	    //Übertragung in Melde-DB
	    "FC63_DB_Copy"(DB_src := 80,
	                   DB_src_offs := 96,
	                   DB_dest := 100,
	                   DB_dest_offs := 64,
	                   count := 34);
	    //div. Messwerte
	    "ZEN_MW".BB_G1_KS_Druck_Netz := INT_TO_REAL("DB80_Peri_EA".Kaeser_G1.E.Druck_Netz) / 1.0;
	    "ZEN_MW".BB_G1_KS_Temp_Verdicht := INT_TO_REAL("DB80_Peri_EA".Kaeser_G1.E.Temp_Verdicht) / 10.0;
	    "ZEN_MW".BB_G1_KS_Temp_Schallhaube := INT_TO_REAL("DB80_Peri_EA".Kaeser_G1.E.Temp_Schallhaube) / 10.0;
	    "ZEN_MW".BB_G1_KS_Temp_Ansaug := INT_TO_REAL("DB80_Peri_EA".Kaeser_G1.E.Temp_Ansaug) / 10.0;
	    "ZEN_MW".BB_G1_KS_Temp_Oel := INT_TO_REAL("DB80_Peri_EA".Kaeser_G1.E.Temp_Oel) / 10.0;
	    "ZEN_MW".BB_G1_KS_Temp_Wicklung := INT_TO_REAL("DB80_Peri_EA".Kaeser_G1.E.Temp_Wicklung) / 10.0;
	    "ZEN_MW".BB_G1_KS_Volumenstrom := INT_TO_REAL("DB80_Peri_EA".Kaeser_G1.E.Volumenstrom) * 6.0;
	    "ZEN_MW".BB_G1_KS_Motorfrequenz := INT_TO_REAL("DB80_Peri_EA".Kaeser_G1.E.Motorfrequenz) / 1.0;
	    "ZEN_MW".BB_G1_KS_Motordrehzahl := UINT_TO_REAL("DB80_Peri_EA".Kaeser_G1.E.Motordrehzahl) / 1.0;
	    "ZEN_MW".BB_G1_KS_Blockdrehzahl := UINT_TO_REAL("DB80_Peri_EA".Kaeser_G1.E.Blockdrehzahl) / 1.0;
	END_IF;
	//dezentrale Peripherie Kaeser Gebläse 2 - Teilnehmer 7
	IF "DB91_DP_aktiv".Tln[7] THEN
	    "FC63_DB_Copy"(DB_src := 0,
	                   DB_src_offs := 1200,
	                   DB_dest := 80,
	                   DB_dest_offs := 296,
	                   count := 128);
	    "FC63_DB_Copy"(DB_src := 80,
	                   DB_src_offs := 424,
	                   DB_dest := 0,
	                   DB_dest_offs := 1200,
	                   count := 64);

	    //Übertragung in Melde-DB
	    "FC63_DB_Copy"(DB_src := 80,
	                   DB_src_offs := 296,
	                   DB_dest := 100,
	                   DB_dest_offs := 98,
	                   count := 34);
	    //div. Messwerte
	    "ZEN_MW".BB_G2_KS_Druck_Netz := INT_TO_REAL("DB80_Peri_EA".Kaeser_G2.E.Druck_Netz) / 1.0;
	    "ZEN_MW".BB_G2_KS_Temp_Verdicht := INT_TO_REAL("DB80_Peri_EA".Kaeser_G2.E.Temp_Verdicht) / 10.0;
	    "ZEN_MW".BB_G2_KS_Temp_Schallhaube := INT_TO_REAL("DB80_Peri_EA".Kaeser_G2.E.Temp_Schallhaube) / 10.0;
	    "ZEN_MW".BB_G2_KS_Temp_Ansaug := INT_TO_REAL("DB80_Peri_EA".Kaeser_G2.E.Temp_Ansaug) / 10.0;
	    "ZEN_MW".BB_G2_KS_Temp_Oel := INT_TO_REAL("DB80_Peri_EA".Kaeser_G2.E.Temp_Oel) / 10.0;
	    "ZEN_MW".BB_G2_KS_Temp_Wicklung := INT_TO_REAL("DB80_Peri_EA".Kaeser_G2.E.Temp_Wicklung) / 10.0;
	    "ZEN_MW".BB_G2_KS_Volumenstrom := INT_TO_REAL("DB80_Peri_EA".Kaeser_G2.E.Volumenstrom) * 6.0;
	    "ZEN_MW".BB_G2_KS_Motorfrequenz := INT_TO_REAL("DB80_Peri_EA".Kaeser_G2.E.Motorfrequenz) / 1.0;
	    "ZEN_MW".BB_G2_KS_Motordrehzahl := UINT_TO_REAL("DB80_Peri_EA".Kaeser_G2.E.Motordrehzahl) / 1.0;
	    "ZEN_MW".BB_G2_KS_Blockdrehzahl := UINT_TO_REAL("DB80_Peri_EA".Kaeser_G2.E.Blockdrehzahl) / 1.0;

	END_IF;
	//dezentrale Peripherie Kaeser Gebläse 3 - Teilnehmer 8
	IF "DB91_DP_aktiv".Tln[8] THEN
	    "FC63_DB_Copy"(DB_src := 0,
	                   DB_src_offs := 1400,
	                   DB_dest := 80,
	                   DB_dest_offs := 496,
	                   count := 128);
	    "FC63_DB_Copy"(DB_src := 80,
	                   DB_src_offs := 624,
	                   DB_dest := 0,
	                   DB_dest_offs := 1400,
	                   count := 64);

	    //Übertragung in Melde-DB
	    "FC63_DB_Copy"(DB_src := 80,
	                   DB_src_offs := 496,
	                   DB_dest := 100,
	                   DB_dest_offs := 132,
	                   count := 34);
	    //div. Messwerte
	    "ZEN_MW".BB_G3_KS_Druck_Netz := INT_TO_REAL("DB80_Peri_EA".Kaeser_G3.E.Druck_Netz) / 1.0;
	    "ZEN_MW".BB_G3_KS_Temp_Verdicht := INT_TO_REAL("DB80_Peri_EA".Kaeser_G3.E.Temp_Verdicht) / 10.0;
	    "ZEN_MW".BB_G3_KS_Temp_Schallhaube := INT_TO_REAL("DB80_Peri_EA".Kaeser_G3.E.Temp_Schallhaube) / 10.0;
	    "ZEN_MW".BB_G3_KS_Temp_Ansaug := INT_TO_REAL("DB80_Peri_EA".Kaeser_G3.E.Temp_Ansaug) / 10.0;
	    "ZEN_MW".BB_G3_KS_Temp_Oel := INT_TO_REAL("DB80_Peri_EA".Kaeser_G3.E.Temp_Oel) / 10.0;
	    "ZEN_MW".BB_G3_KS_Temp_Wicklung := INT_TO_REAL("DB80_Peri_EA".Kaeser_G3.E.Temp_Wicklung) / 10.0;
	    "ZEN_MW".BB_G3_KS_Volumenstrom := INT_TO_REAL("DB80_Peri_EA".Kaeser_G3.E.Volumenstrom)*6.0;
	    "ZEN_MW".BB_G3_KS_Motorfrequenz := INT_TO_REAL("DB80_Peri_EA".Kaeser_G3.E.Motorfrequenz) / 1.0;
	    "ZEN_MW".BB_G3_KS_Motordrehzahl := UINT_TO_REAL("DB80_Peri_EA".Kaeser_G3.E.Motordrehzahl) / 1.0;
	    "ZEN_MW".BB_G3_KS_Blockdrehzahl := UINT_TO_REAL("DB80_Peri_EA".Kaeser_G3.E.Blockdrehzahl) / 1.0;

	END_IF;


	"ZEN_Meld".ZEN_DiagKom_DP_BF3 := NOT "DB91_DP_aktiv".Tln[3];
	"ZEN_Meld".ZEN_DiagKom_DP_BF4 := NOT "DB91_DP_aktiv".Tln[4];
	"ZEN_Meld".ZEN_DiagKom_DP_BF5 := NOT "DB91_DP_aktiv".Tln[5];
	"ZEN_Meld".ZEN_DiagKom_DP_BF6 := NOT "DB91_DP_aktiv".Tln[6];
	"ZEN_Meld".ZEN_DiagKom_DP_BF7 := NOT "DB91_DP_aktiv".Tln[7];
	"ZEN_Meld".ZEN_DiagKom_DP_BF8 := NOT "DB91_DP_aktiv".Tln[8];
	"ZEN_Meld".ZEN_DiagKom_DP_BF10 := NOT "DB91_DP_aktiv".Tln[10];

	//Meldungen für OP
	//
	IF 1 THEN

	    "DB92_OP_Data".Msg_B0[0].%X0 := "ZEN_Meld".E_Zulauf_AR_P1_St;
	    "DB92_OP_Data".Msg_B0[0].%X1 := "ZEN_Meld".E_Zulauf_AR_SS;
	    "DB92_OP_Data".Msg_B0[0].%X2 := "ZEN_Meld".E_Zulauf_AR_P2_St;
	    "DB92_OP_Data".Msg_B0[0].%X3 := "ZEN_Meld".E_Zulauf_AR_HW;
	    "DB92_OP_Data".Msg_B0[0].%X4 := "ZEN_Meld".E_Zulauf_AR_Niv_St;
	    "DB92_OP_Data".Msg_B0[0].%X5 := "ZEN_Meld".E_Zulauf_AR_DF_St;
	    "DB92_OP_Data".Msg_B0[0].%X6 := "ZEN_Meld".E_Ablauf_pH_St;
	    "DB92_OP_Data".Msg_B0[0].%X7 := "ZEN_Meld".E_Ablauf_O2_St;
	    "DB92_OP_Data".Msg_B0[0].%X8 := "ZEN_Meld".E_Ablauf_DF_St;
	    "DB92_OP_Data".Msg_B0[0].%X9 := "ZEN_Meld".E_NSHV_SS1_St;
	    "DB92_OP_Data".Msg_B0[0].%X10 := "ZEN_Meld".E_NSHV_SS2_St;
	    "DB92_OP_Data".Msg_B0[0].%X11 := "ZEN_Meld".E_NSHV_N02_AF_St;
	    "DB92_OP_Data".Msg_B0[0].%X12 := "ZEN_Meld".E_NSHV_N03_AF_St;
	    "DB92_OP_Data".Msg_B0[0].%X13 := "ZEN_Meld".E_NSHV_N04_AF_St;
	    "DB92_OP_Data".Msg_B0[0].%X14 := "ZEN_Meld".E_NSHV_LS_Aus;
	    "DB92_OP_Data".Msg_B0[0].%X15 := "ZEN_Meld".E_NSHV_LS_St;
	    "DB92_OP_Data".Msg_B0[1].%X0 := "ZEN_Meld".E_NSHV_NA;
	    "DB92_OP_Data".Msg_B0[1].%X1 := "ZEN_Meld".E_BB_G1_St;
	    "DB92_OP_Data".Msg_B0[1].%X2 := "ZEN_Meld".E_BB_G1_AF_St;
	    "DB92_OP_Data".Msg_B0[1].%X3 := "ZEN_Meld".E_BB_SHL_G1_St;
	    "DB92_OP_Data".Msg_B0[1].%X4 := "ZEN_Meld".E_BB_G2_St;
	    "DB92_OP_Data".Msg_B0[1].%X5 := "ZEN_Meld".E_BB_G2_AF_St;
	    "DB92_OP_Data".Msg_B0[1].%X6 := "ZEN_Meld".E_BB_SHL_G2_St;
	    "DB92_OP_Data".Msg_B0[1].%X7 := "ZEN_Meld".E_BB_G3_St;
	    "DB92_OP_Data".Msg_B0[1].%X8 := "ZEN_Meld".E_BB_G3_AF_St;
	    "DB92_OP_Data".Msg_B0[1].%X9 := "ZEN_Meld".E_BB_SHL_G3_St;
	    "DB92_OP_Data".Msg_B0[1].%X10 := "ZEN_Meld".E_BB_AV_St;
	    "DB92_OP_Data".Msg_B0[1].%X11 := "ZEN_Meld".E_BB_AV_AF_St;
	    "DB92_OP_Data".Msg_B0[1].%X12 := "ZEN_Meld".E_BB_RT;
	    "DB92_OP_Data".Msg_B0[1].%X13 := "ZEN_Meld".E_BB1_SR_K_St;
	    "DB92_OP_Data".Msg_B0[1].%X14 := "ZEN_Meld".E_BB1_SR_K_AF_St;
	    "DB92_OP_Data".Msg_B0[1].%X15 := "ZEN_Meld".E_BB_LS1_St;
	    "DB92_OP_Data".Msg_B0[2].%X0 := "ZEN_Meld".E_BB_LS1_AF_St;
	    "DB92_OP_Data".Msg_B0[2].%X1 := "ZEN_Meld".E_BB_LS2_St;
	    "DB92_OP_Data".Msg_B0[2].%X2 := "ZEN_Meld".E_BB_LS2_AF_St;
	    "DB92_OP_Data".Msg_B0[2].%X3 := "ZEN_Meld".E_BB1_RZP1_St;
	    "DB92_OP_Data".Msg_B0[2].%X4 := "ZEN_Meld".E_BB1_RZP1_AF_St;
	    "DB92_OP_Data".Msg_B0[2].%X5 := "ZEN_Meld".E_BB1_RZP2_St;
	    "DB92_OP_Data".Msg_B0[2].%X6 := "ZEN_Meld".E_BB1_RZP2_AF_St;
	    "DB92_OP_Data".Msg_B0[2].%X7 := "ZEN_Meld".E_BB1_UeSP_St;
	    "DB92_OP_Data".Msg_B0[2].%X8 := "ZEN_Meld".E_BB1_UeSP_AF_St;
	    "DB92_OP_Data".Msg_B0[2].%X9 := "ZEN_Meld".E_BB1_AS1_St;
	    "DB92_OP_Data".Msg_B0[2].%X10 := "ZEN_Meld".E_BB1_AS1_AF_St;
	    "DB92_OP_Data".Msg_B0[2].%X11 := "ZEN_Meld".E_BB1_AS2_St;
	    "DB92_OP_Data".Msg_B0[2].%X12 := "ZEN_Meld".E_BB1_AS2_AF_St;
	    "DB92_OP_Data".Msg_B0[2].%X13 := "ZEN_Meld".E_BB1_SR1_AF_St;
	    "DB92_OP_Data".Msg_B0[2].%X14 := "ZEN_Meld".E_BB1_SR2_AF_St;
	    "DB92_OP_Data".Msg_B0[2].%X15 := "ZEN_Meld".E_BB1_O2_St;
	    "DB92_OP_Data".Msg_B0[3].%X0 := "ZEN_Meld".E_BB1_DF_St;
	    "DB92_OP_Data".Msg_B0[3].%X1 := "ZEN_Meld".E_BB2_RZP1_St;
	    "DB92_OP_Data".Msg_B0[3].%X2 := "ZEN_Meld".E_BB2_RZP1_AF_St;
	    "DB92_OP_Data".Msg_B0[3].%X3 := "ZEN_Meld".E_BB2_RZP2_St;
	    "DB92_OP_Data".Msg_B0[3].%X4 := "ZEN_Meld".E_BB2_RZP2_AF_St;
	    "DB92_OP_Data".Msg_B0[3].%X5 := "ZEN_Meld".E_BB2_UeSP_St;
	    "DB92_OP_Data".Msg_B0[3].%X6 := "ZEN_Meld".E_BB2_UeSP_AF_St;
	    "DB92_OP_Data".Msg_B0[3].%X7 := "ZEN_Meld".E_BB2_AS1_St;
	    "DB92_OP_Data".Msg_B0[3].%X8 := "ZEN_Meld".E_BB2_AS1_AF_St;
	    "DB92_OP_Data".Msg_B0[3].%X9 := "ZEN_Meld".E_BB2_AS2_St;
	    "DB92_OP_Data".Msg_B0[3].%X10 := "ZEN_Meld".E_BB2_AS2_AF_St;
	    "DB92_OP_Data".Msg_B0[3].%X11 := "ZEN_Meld".E_BB2_SR1_AF_St;
	    "DB92_OP_Data".Msg_B0[3].%X12 := "ZEN_Meld".E_BB2_SR2_AF_St;
	    "DB92_OP_Data".Msg_B0[3].%X13 := "ZEN_Meld".E_BB2_O2_St;
	    "DB92_OP_Data".Msg_B0[3].%X14 := "ZEN_Meld".E_BB2_DF_St;
	    "DB92_OP_Data".Msg_B0[3].%X15 := "ZEN_Meld".E_BB2_SR_K_St;
	    "DB92_OP_Data".Msg_B0[4].%X0 := "ZEN_Meld".E_BB2_SR_K_AF_St;
	    "DB92_OP_Data".Msg_B0[4].%X1 := "ZEN_Meld".E_Zulauf_RA_SA_St;
	    "DB92_OP_Data".Msg_B0[4].%X2 := "ZEN_Meld".E_Zulauf_RA_HZS_St;
	    "DB92_OP_Data".Msg_B0[4].%X3 := "ZEN_Meld".E_Zulauf_RA_VKS_St;
	    "DB92_OP_Data".Msg_B0[4].%X4 := "ZEN_Meld".E_Zulauf_RA_V_St;
	    "DB92_OP_Data".Msg_B0[4].%X5 := "ZEN_Meld".E_Zulauf_RA_RP_St;
	    "DB92_OP_Data".Msg_B0[4].%X6 := "ZEN_Meld".E_Zulauf_RA_FP_St;
	    "DB92_OP_Data".Msg_B0[4].%X7 := "ZEN_Meld".E_Zulauf_RA_24V_St;
	    "DB92_OP_Data".Msg_B0[4].%X8 := "ZEN_Meld".E_Zulauf_RA_US_St;
	    "DB92_OP_Data".Msg_B0[4].%X9 := "ZEN_Meld".E_Zulauf_RA_230V_St;
	    "DB92_OP_Data".Msg_B0[4].%X10 := "ZEN_Meld".E_Zulauf_DF_St;
	    "DB92_OP_Data".Msg_B0[4].%X11 := "ZEN_Meld".E_Zulauf_Niv_St;
	    "DB92_OP_Data".Msg_B0[4].%X12 := "ZEN_Meld".E_Verteiler_pH_St;
	    "DB92_OP_Data".Msg_B0[4].%X13 := "ZEN_Meld".E_Zulauf_AS_St;
	    "DB92_OP_Data".Msg_B0[4].%X14 := "ZEN_Meld".E_Zulauf_AS_AF_St;
	    "DB92_OP_Data".Msg_B0[4].%X15 := "ZEN_Meld".E_Schlamm_BP_St;
	    "DB92_OP_Data".Msg_B0[5].%X0 := "ZEN_Meld".E_Schlamm_BP_AF_St;
	    "DB92_OP_Data".Msg_B0[5].%X1 := "ZEN_Meld".E_Truebwasser_P1_St;
	    "DB92_OP_Data".Msg_B0[5].%X2 := "ZEN_Meld".E_Truebwasser_P1_AF_St;
	    "DB92_OP_Data".Msg_B0[5].%X3 := "ZEN_Meld".E_Truebwasser_P2_St;
	    "DB92_OP_Data".Msg_B0[5].%X4 := "ZEN_Meld".E_Truebwasser_P2_AF_St;
	    "DB92_OP_Data".Msg_B0[5].%X5 := "ZEN_Meld".E_Schlamm_AS_St;
	    "DB92_OP_Data".Msg_B0[5].%X6 := "ZEN_Meld".E_Schlamm_AS_AF_St;
	    "DB92_OP_Data".Msg_B0[5].%X7 := "ZEN_Meld".E_Schlamm_Besch_DF_St;
	    "DB92_OP_Data".Msg_B0[5].%X8 := "ZEN_Meld".E_Truebwasser_Niv_St;
	    "DB92_OP_Data".Msg_B0[5].%X9 := "ZEN_Meld".E_Truebwasser_DF_St;
	    "DB92_OP_Data".Msg_B0[5].%X10 := "ZEN_Meld".ZEN_DiagKom_IEC;
	    "DB92_OP_Data".Msg_B0[5].%X11 := "ZEN_Meld".ZEN_DiagKom_DP_BF3;
	    "DB92_OP_Data".Msg_B0[5].%X12 := "ZEN_Meld".ZEN_DiagKom_DP_BF4;
	    "DB92_OP_Data".Msg_B0[5].%X13 := "ZEN_Meld".ZEN_ObjS_Alarm;
	    "DB92_OP_Data".Msg_B0[5].%X14 := "ZEN_Meld".ZEN_ObjS_unscharf;
	    "DB92_OP_Data".Msg_B0[5].%X15 := "ZEN_Meld".ZEN_NA_res;
	    "DB92_OP_Data".Msg_B0[6].%X0 := "ZEN_Meld".Biocos1_Auto_Bel_O2_St;
	    "DB92_OP_Data".Msg_B0[6].%X1 := "ZEN_Meld".Biocos1_Auto_Bel_O2_min;
	    "DB92_OP_Data".Msg_B0[6].%X2 := "ZEN_Meld".Biocos1_Auto_UeSS_Menge_St;
	    "DB92_OP_Data".Msg_B0[6].%X3 := "ZEN_Meld".Biocos2_Auto_Bel_O2_St;
	    "DB92_OP_Data".Msg_B0[6].%X4 := "ZEN_Meld".Biocos2_Auto_Bel_O2_min;
	    "DB92_OP_Data".Msg_B0[6].%X5 := "ZEN_Meld".Biocos2_Auto_UeSS_Menge_St;
	    "DB92_OP_Data".Msg_B0[6].%X6 := "ZEN_Meld".Zulauf_PW_Auto_DF_max;
	    "DB92_OP_Data".Msg_B0[6].%X7 := "ZEN_Meld".Zulauf_PW_Auto_Niv_max;
	    "DB92_OP_Data".Msg_B0[6].%X8 := "ZEN_Meld".Zulauf_PW_Auto_Niv_AS;
	    "DB92_OP_Data".Msg_B0[6].%X9 := "ZEN_Meld".Zulauf_PW_Auto_Frg_Aus;
	    "DB92_OP_Data".Msg_B0[6].%X10 := "ZEN_Meld".Zulauf_RA_SA_Stillst;
	    "DB92_OP_Data".Msg_B0[6].%X11 := "ZEN_Meld".Schlamm_Besch_Auto_Zt_max;
	    "DB92_OP_Data".Msg_B0[6].%X12 := "DB104_Antriebe_Meld".BB_G1.Stoerung.Wa_EZ;
	    "DB92_OP_Data".Msg_B0[6].%X13 := "DB104_Antriebe_Meld".BB_G1.Stoerung.Wa_Wart;
	    "DB92_OP_Data".Msg_B0[6].%X14 := "DB104_Antriebe_Meld".BB_G2.Stoerung.Wa_EZ;
	    "DB92_OP_Data".Msg_B0[6].%X15 := "DB104_Antriebe_Meld".BB_G2.Stoerung.Wa_Wart;
	    "DB92_OP_Data".Msg_B0[7].%X0 := "DB104_Antriebe_Meld".BB_G3.Stoerung.Wa_EZ;
	    "DB92_OP_Data".Msg_B0[7].%X1 := "DB104_Antriebe_Meld".BB_G3.Stoerung.Wa_Wart;
	    "DB92_OP_Data".Msg_B0[7].%X2 := "DB104_Antriebe_Meld".BB_SHL_G1.Stoerung.Wa_EZ;
	    "DB92_OP_Data".Msg_B0[7].%X3 := "DB104_Antriebe_Meld".BB_SHL_G1.Stoerung.Wa_Wart;
	    "DB92_OP_Data".Msg_B0[7].%X4 := "DB104_Antriebe_Meld".BB_SHL_G2.Stoerung.Wa_EZ;
	    "DB92_OP_Data".Msg_B0[7].%X5 := "DB104_Antriebe_Meld".BB_SHL_G2.Stoerung.Wa_Wart;
	    "DB92_OP_Data".Msg_B0[7].%X6 := "DB104_Antriebe_Meld".BB_SHL_G3.Stoerung.Wa_EZ;
	    "DB92_OP_Data".Msg_B0[7].%X7 := "DB104_Antriebe_Meld".BB_SHL_G3.Stoerung.Wa_Wart;
	    "DB92_OP_Data".Msg_B0[7].%X8 := "DB104_Antriebe_Meld".BB_AV.Stoerung.Wa_EZ;
	    "DB92_OP_Data".Msg_B0[7].%X9 := "DB104_Antriebe_Meld".BB_AV.Stoerung.Wa_Wart;
	    "DB92_OP_Data".Msg_B0[7].%X10 := "DB104_Antriebe_Meld".BB_LS1.Stoerung.Wa_EZ;
	    "DB92_OP_Data".Msg_B0[7].%X11 := "DB104_Antriebe_Meld".BB_LS1.Stoerung.Wa_Wart;
	    "DB92_OP_Data".Msg_B0[7].%X12 := "DB104_Antriebe_Meld".BB_LS2.Stoerung.Wa_EZ;
	    "DB92_OP_Data".Msg_B0[7].%X13 := "DB104_Antriebe_Meld".BB_LS2.Stoerung.Wa_Wart;
	    "DB92_OP_Data".Msg_B0[7].%X14 := "DB104_Antriebe_Meld".BB1_RZP1.Stoerung.Wa_EZ;
	    "DB92_OP_Data".Msg_B0[7].%X15 := "DB104_Antriebe_Meld".BB1_RZP1.Stoerung.Wa_Wart;
	    "DB92_OP_Data".Msg_B0[8].%X0 := "DB104_Antriebe_Meld".BB1_RZP2.Stoerung.Wa_EZ;
	    "DB92_OP_Data".Msg_B0[8].%X1 := "DB104_Antriebe_Meld".BB1_RZP2.Stoerung.Wa_Wart;
	    "DB92_OP_Data".Msg_B0[8].%X2 := "DB104_Antriebe_Meld".BB1_UeSP.Stoerung.Wa_EZ;
	    "DB92_OP_Data".Msg_B0[8].%X3 := "DB104_Antriebe_Meld".BB1_UeSP.Stoerung.Wa_Wart;
	    "DB92_OP_Data".Msg_B0[8].%X4 := "DB104_Antriebe_Meld".BB1_AS1.Stoerung.Wa_EZ;
	    "DB92_OP_Data".Msg_B0[8].%X5 := "DB104_Antriebe_Meld".BB1_AS1.Stoerung.Wa_Wart;
	    "DB92_OP_Data".Msg_B0[8].%X6 := "DB104_Antriebe_Meld".BB1_AS2.Stoerung.Wa_EZ;
	    "DB92_OP_Data".Msg_B0[8].%X7 := "DB104_Antriebe_Meld".BB1_AS2.Stoerung.Wa_Wart;
	    "DB92_OP_Data".Msg_B0[8].%X8 := "DB104_Antriebe_Meld".BB1_SR1.Stoerung.Wa_EZ;
	    "DB92_OP_Data".Msg_B0[8].%X9 := "DB104_Antriebe_Meld".BB1_SR1.Stoerung.Wa_Wart;
	    "DB92_OP_Data".Msg_B0[8].%X10 := "DB104_Antriebe_Meld".BB1_SR2.Stoerung.Wa_EZ;
	    "DB92_OP_Data".Msg_B0[8].%X11 := "DB104_Antriebe_Meld".BB1_SR2.Stoerung.Wa_Wart;
	    "DB92_OP_Data".Msg_B0[8].%X12 := "DB104_Antriebe_Meld".BB2_RZP1.Stoerung.Wa_EZ;
	    "DB92_OP_Data".Msg_B0[8].%X13 := "DB104_Antriebe_Meld".BB2_RZP1.Stoerung.Wa_Wart;
	    "DB92_OP_Data".Msg_B0[8].%X14 := "DB104_Antriebe_Meld".BB2_RZP2.Stoerung.Wa_EZ;
	    "DB92_OP_Data".Msg_B0[8].%X15 := "DB104_Antriebe_Meld".BB2_RZP2.Stoerung.Wa_Wart;
	    "DB92_OP_Data".Msg_B0[9].%X0 := "DB104_Antriebe_Meld".BB2_UeSP.Stoerung.Wa_EZ;
	    "DB92_OP_Data".Msg_B0[9].%X1 := "DB104_Antriebe_Meld".BB2_UeSP.Stoerung.Wa_Wart;
	    "DB92_OP_Data".Msg_B0[9].%X2 := "DB104_Antriebe_Meld".BB2_AS1.Stoerung.Wa_EZ;
	    "DB92_OP_Data".Msg_B0[9].%X3 := "DB104_Antriebe_Meld".BB2_AS1.Stoerung.Wa_Wart;
	    "DB92_OP_Data".Msg_B0[9].%X4 := "DB104_Antriebe_Meld".BB2_AS2.Stoerung.Wa_EZ;
	    "DB92_OP_Data".Msg_B0[9].%X5 := "DB104_Antriebe_Meld".BB2_AS2.Stoerung.Wa_Wart;
	    "DB92_OP_Data".Msg_B0[9].%X6 := "DB104_Antriebe_Meld".BB2_SR1.Stoerung.Wa_EZ;
	    "DB92_OP_Data".Msg_B0[9].%X7 := "DB104_Antriebe_Meld".BB2_SR1.Stoerung.Wa_Wart;
	    "DB92_OP_Data".Msg_B0[9].%X8 := "DB104_Antriebe_Meld".BB2_SR2.Stoerung.Wa_EZ;
	    "DB92_OP_Data".Msg_B0[9].%X9 := "DB104_Antriebe_Meld".BB2_SR2.Stoerung.Wa_Wart;
	    "DB92_OP_Data".Msg_B0[9].%X10 := "DB104_Antriebe_Meld".Zulauf_AR_P1.Stoerung.Wa_EZ;
	    "DB92_OP_Data".Msg_B0[9].%X11 := "DB104_Antriebe_Meld".Zulauf_AR_P1.Stoerung.Wa_Wart;
	    "DB92_OP_Data".Msg_B0[9].%X12 := "DB104_Antriebe_Meld".Zulauf_AR_P2.Stoerung.Wa_EZ;
	    "DB92_OP_Data".Msg_B0[9].%X13 := "DB104_Antriebe_Meld".Zulauf_AR_P2.Stoerung.Wa_Wart;
	    "DB92_OP_Data".Msg_B0[9].%X14 := "DB104_Antriebe_Meld".Zulauf_AS.Stoerung.Wa_EZ;
	    "DB92_OP_Data".Msg_B0[9].%X15 := "DB104_Antriebe_Meld".Zulauf_AS.Stoerung.Wa_Wart;
	    "DB92_OP_Data".Msg_B0[10].%X0 := "DB104_Antriebe_Meld".Zulauf_RA_SA.Stoerung.Wa_EZ;
	    "DB92_OP_Data".Msg_B0[10].%X1 := "DB104_Antriebe_Meld".Zulauf_RA_SA.Stoerung.Wa_Wart;
	    "DB92_OP_Data".Msg_B0[10].%X2 := "DB104_Antriebe_Meld".Zulauf_RA_HZS.Stoerung.Wa_EZ;
	    "DB92_OP_Data".Msg_B0[10].%X3 := "DB104_Antriebe_Meld".Zulauf_RA_HZS.Stoerung.Wa_Wart;
	    "DB92_OP_Data".Msg_B0[10].%X4 := "DB104_Antriebe_Meld".Zulauf_RA_VKS.Stoerung.Wa_EZ;
	    "DB92_OP_Data".Msg_B0[10].%X5 := "DB104_Antriebe_Meld".Zulauf_RA_VKS.Stoerung.Wa_Wart;
	    "DB92_OP_Data".Msg_B0[10].%X6 := "DB104_Antriebe_Meld".Zulauf_RA_V.Stoerung.Wa_EZ;
	    "DB92_OP_Data".Msg_B0[10].%X7 := "DB104_Antriebe_Meld".Zulauf_RA_V.Stoerung.Wa_Wart;
	    "DB92_OP_Data".Msg_B0[10].%X8 := "DB104_Antriebe_Meld".Zulauf_RA_RP.Stoerung.Wa_EZ;
	    "DB92_OP_Data".Msg_B0[10].%X9 := "DB104_Antriebe_Meld".Zulauf_RA_RP.Stoerung.Wa_Wart;
	    "DB92_OP_Data".Msg_B0[10].%X10 := "DB104_Antriebe_Meld".Zulauf_RA_FP.Stoerung.Wa_EZ;
	    "DB92_OP_Data".Msg_B0[10].%X11 := "DB104_Antriebe_Meld".Zulauf_RA_FP.Stoerung.Wa_Wart;
	    "DB92_OP_Data".Msg_B0[10].%X12 := "DB104_Antriebe_Meld".Schlamm_BP.Stoerung.Wa_EZ;
	    "DB92_OP_Data".Msg_B0[10].%X13 := "DB104_Antriebe_Meld".Schlamm_BP.Stoerung.Wa_Wart;
	    "DB92_OP_Data".Msg_B0[10].%X14 := "DB104_Antriebe_Meld".Truebwasser_P1.Stoerung.Wa_EZ;
	    "DB92_OP_Data".Msg_B0[10].%X15 := "DB104_Antriebe_Meld".Truebwasser_P1.Stoerung.Wa_Wart;
	    "DB92_OP_Data".Msg_B0[11].%X0 := "DB104_Antriebe_Meld".Truebwasser_P2.Stoerung.Wa_EZ;
	    "DB92_OP_Data".Msg_B0[11].%X1 := "DB104_Antriebe_Meld".Truebwasser_P2.Stoerung.Wa_Wart;
	    "DB92_OP_Data".Msg_B0[11].%X2 := "DB104_Antriebe_Meld".Schlamm_AS.Stoerung.Wa_EZ;
	    "DB92_OP_Data".Msg_B0[11].%X3 := "DB104_Antriebe_Meld".Schlamm_AS.Stoerung.Wa_Wart;
	    "DB92_OP_Data".Msg_B0[11].%X4 := "DB114_MW_Meld".Zulauf_AR_Niv.Stoerung.GW_HH;
	    "DB92_OP_Data".Msg_B0[11].%X5 := "DB114_MW_Meld".Zulauf_AR_Niv.Stoerung.GW_H;
	    "DB92_OP_Data".Msg_B0[11].%X6 := "DB114_MW_Meld".Zulauf_AR_Niv.Stoerung.GW_L;
	    "DB92_OP_Data".Msg_B0[11].%X7 := "DB114_MW_Meld".Zulauf_AR_Niv.Stoerung.GW_LL;
	    "DB92_OP_Data".Msg_B0[11].%X8 := "DB114_MW_Meld".Zulauf_AR_Temp.Stoerung.GW_HH;
	    "DB92_OP_Data".Msg_B0[11].%X9 := "DB114_MW_Meld".Zulauf_AR_Temp.Stoerung.GW_H;
	    "DB92_OP_Data".Msg_B0[11].%X10 := "DB114_MW_Meld".Zulauf_AR_Temp.Stoerung.GW_L;
	    "DB92_OP_Data".Msg_B0[11].%X11 := "DB114_MW_Meld".Zulauf_AR_Temp.Stoerung.GW_LL;
	    "DB92_OP_Data".Msg_B0[11].%X12 := "DB114_MW_Meld".Zulauf_AR_DF.Stoerung.GW_HH;
	    "DB92_OP_Data".Msg_B0[11].%X13 := "DB114_MW_Meld".Zulauf_AR_DF.Stoerung.GW_H;
	    "DB92_OP_Data".Msg_B0[11].%X14 := "DB114_MW_Meld".Zulauf_AR_DF.Stoerung.GW_L;
	    "DB92_OP_Data".Msg_B0[11].%X15 := "DB114_MW_Meld".Zulauf_AR_DF.Stoerung.GW_LL;
	    "DB92_OP_Data".Msg_B0[12].%X0 := "DB114_MW_Meld".BB1_AS1_SS.Stoerung.GW_HH;
	    "DB92_OP_Data".Msg_B0[12].%X1 := "DB114_MW_Meld".BB1_AS1_SS.Stoerung.GW_H;
	    "DB92_OP_Data".Msg_B0[12].%X2 := "DB114_MW_Meld".BB1_AS1_SS.Stoerung.GW_L;
	    "DB92_OP_Data".Msg_B0[12].%X3 := "DB114_MW_Meld".BB1_AS1_SS.Stoerung.GW_LL;
	    "DB92_OP_Data".Msg_B0[12].%X4 := "DB114_MW_Meld".BB1_AS2_SS.Stoerung.GW_HH;
	    "DB92_OP_Data".Msg_B0[12].%X5 := "DB114_MW_Meld".BB1_AS2_SS.Stoerung.GW_H;
	    "DB92_OP_Data".Msg_B0[12].%X6 := "DB114_MW_Meld".BB1_AS2_SS.Stoerung.GW_L;
	    "DB92_OP_Data".Msg_B0[12].%X7 := "DB114_MW_Meld".BB1_AS2_SS.Stoerung.GW_LL;
	    "DB92_OP_Data".Msg_B0[12].%X8 := "DB114_MW_Meld".BB2_AS1_SS.Stoerung.GW_HH;
	    "DB92_OP_Data".Msg_B0[12].%X9 := "DB114_MW_Meld".BB2_AS1_SS.Stoerung.GW_H;
	    "DB92_OP_Data".Msg_B0[12].%X10 := "DB114_MW_Meld".BB2_AS1_SS.Stoerung.GW_L;
	    "DB92_OP_Data".Msg_B0[12].%X11 := "DB114_MW_Meld".BB2_AS1_SS.Stoerung.GW_LL;
	    "DB92_OP_Data".Msg_B0[12].%X12 := "DB114_MW_Meld".BB2_AS2_SS.Stoerung.GW_HH;
	    "DB92_OP_Data".Msg_B0[12].%X13 := "DB114_MW_Meld".BB2_AS2_SS.Stoerung.GW_H;
	    "DB92_OP_Data".Msg_B0[12].%X14 := "DB114_MW_Meld".BB2_AS2_SS.Stoerung.GW_L;
	    "DB92_OP_Data".Msg_B0[12].%X15 := "DB114_MW_Meld".BB2_AS2_SS.Stoerung.GW_LL;
	    "DB92_OP_Data".Msg_B0[13].%X0 := "DB114_MW_Meld".BB1_O2.Stoerung.GW_HH;
	    "DB92_OP_Data".Msg_B0[13].%X1 := "DB114_MW_Meld".BB1_O2.Stoerung.GW_H;
	    "DB92_OP_Data".Msg_B0[13].%X2 := "DB114_MW_Meld".BB1_O2.Stoerung.GW_L;
	    "DB92_OP_Data".Msg_B0[13].%X3 := "DB114_MW_Meld".BB1_O2.Stoerung.GW_LL;
	    "DB92_OP_Data".Msg_B0[13].%X4 := "DB114_MW_Meld".BB1_Temp.Stoerung.GW_HH;
	    "DB92_OP_Data".Msg_B0[13].%X5 := "DB114_MW_Meld".BB1_Temp.Stoerung.GW_H;
	    "DB92_OP_Data".Msg_B0[13].%X6 := "DB114_MW_Meld".BB1_Temp.Stoerung.GW_L;
	    "DB92_OP_Data".Msg_B0[13].%X7 := "DB114_MW_Meld".BB1_Temp.Stoerung.GW_LL;
	    "DB92_OP_Data".Msg_B0[13].%X8 := "DB114_MW_Meld".BB2_O2.Stoerung.GW_HH;
	    "DB92_OP_Data".Msg_B0[13].%X9 := "DB114_MW_Meld".BB2_O2.Stoerung.GW_H;
	    "DB92_OP_Data".Msg_B0[13].%X10 := "DB114_MW_Meld".BB2_O2.Stoerung.GW_L;
	    "DB92_OP_Data".Msg_B0[13].%X11 := "DB114_MW_Meld".BB2_O2.Stoerung.GW_LL;
	    "DB92_OP_Data".Msg_B0[13].%X12 := "DB114_MW_Meld".BB2_Temp.Stoerung.GW_HH;
	    "DB92_OP_Data".Msg_B0[13].%X13 := "DB114_MW_Meld".BB2_Temp.Stoerung.GW_H;
	    "DB92_OP_Data".Msg_B0[13].%X14 := "DB114_MW_Meld".BB2_Temp.Stoerung.GW_L;
	    "DB92_OP_Data".Msg_B0[13].%X15 := "DB114_MW_Meld".BB2_Temp.Stoerung.GW_LL;
	    "DB92_OP_Data".Msg_B0[14].%X0 := "DB114_MW_Meld".BB1_DF.Stoerung.GW_HH;
	    "DB92_OP_Data".Msg_B0[14].%X1 := "DB114_MW_Meld".BB1_DF.Stoerung.GW_H;
	    "DB92_OP_Data".Msg_B0[14].%X2 := "DB114_MW_Meld".BB1_DF.Stoerung.GW_L;
	    "DB92_OP_Data".Msg_B0[14].%X3 := "DB114_MW_Meld".BB1_DF.Stoerung.GW_LL;
	    "DB92_OP_Data".Msg_B0[14].%X4 := "DB114_MW_Meld".BB2_DF.Stoerung.GW_HH;
	    "DB92_OP_Data".Msg_B0[14].%X5 := "DB114_MW_Meld".BB2_DF.Stoerung.GW_H;
	    "DB92_OP_Data".Msg_B0[14].%X6 := "DB114_MW_Meld".BB2_DF.Stoerung.GW_L;
	    "DB92_OP_Data".Msg_B0[14].%X7 := "DB114_MW_Meld".BB2_DF.Stoerung.GW_LL;
	    "DB92_OP_Data".Msg_B0[14].%X8 := "DB114_MW_Meld".Zulauf_Niv.Stoerung.GW_HH;
	    "DB92_OP_Data".Msg_B0[14].%X9 := "DB114_MW_Meld".Zulauf_Niv.Stoerung.GW_H;
	    "DB92_OP_Data".Msg_B0[14].%X10 := "DB114_MW_Meld".Zulauf_Niv.Stoerung.GW_L;
	    "DB92_OP_Data".Msg_B0[14].%X11 := "DB114_MW_Meld".Zulauf_Niv.Stoerung.GW_LL;
	    "DB92_OP_Data".Msg_B0[14].%X12 := "DB114_MW_Meld".Zulauf_DF.Stoerung.GW_HH;
	    "DB92_OP_Data".Msg_B0[14].%X13 := "DB114_MW_Meld".Zulauf_DF.Stoerung.GW_H;
	    "DB92_OP_Data".Msg_B0[14].%X14 := "DB114_MW_Meld".Zulauf_DF.Stoerung.GW_L;
	    "DB92_OP_Data".Msg_B0[14].%X15 := "DB114_MW_Meld".Zulauf_DF.Stoerung.GW_LL;
	    "DB92_OP_Data".Msg_B0[15].%X0 := "DB114_MW_Meld".Verteiler_pH.Stoerung.GW_HH;
	    "DB92_OP_Data".Msg_B0[15].%X1 := "DB114_MW_Meld".Verteiler_pH.Stoerung.GW_H;
	    "DB92_OP_Data".Msg_B0[15].%X2 := "DB114_MW_Meld".Verteiler_pH.Stoerung.GW_L;
	    "DB92_OP_Data".Msg_B0[15].%X3 := "DB114_MW_Meld".Verteiler_pH.Stoerung.GW_LL;
	    "DB92_OP_Data".Msg_B0[15].%X4 := "DB114_MW_Meld".Verteiler_O2.Stoerung.GW_HH;
	    "DB92_OP_Data".Msg_B0[15].%X5 := "DB114_MW_Meld".Verteiler_O2.Stoerung.GW_H;
	    "DB92_OP_Data".Msg_B0[15].%X6 := "DB114_MW_Meld".Verteiler_O2.Stoerung.GW_L;
	    "DB92_OP_Data".Msg_B0[15].%X7 := "DB114_MW_Meld".Verteiler_O2.Stoerung.GW_LL;
	    "DB92_OP_Data".Msg_B0[15].%X8 := "DB114_MW_Meld".Verteiler_Temp.Stoerung.GW_HH;
	    "DB92_OP_Data".Msg_B0[15].%X9 := "DB114_MW_Meld".Verteiler_Temp.Stoerung.GW_H;
	    "DB92_OP_Data".Msg_B0[15].%X10 := "DB114_MW_Meld".Verteiler_Temp.Stoerung.GW_L;
	    "DB92_OP_Data".Msg_B0[15].%X11 := "DB114_MW_Meld".Verteiler_Temp.Stoerung.GW_LL;
	    "DB92_OP_Data".Msg_B0[15].%X12 := "DB114_MW_Meld".BB_UeSS_DF.Stoerung.GW_HH;
	    "DB92_OP_Data".Msg_B0[15].%X13 := "DB114_MW_Meld".BB_UeSS_DF.Stoerung.GW_H;
	    "DB92_OP_Data".Msg_B0[15].%X14 := "DB114_MW_Meld".BB_UeSS_DF.Stoerung.GW_L;
	    "DB92_OP_Data".Msg_B0[15].%X15 := "DB114_MW_Meld".BB_UeSS_DF.Stoerung.GW_LL;
	    "DB92_OP_Data".Msg_B0[16].%X0 := "DB114_MW_Meld".Ablauf_DF.Stoerung.GW_HH;
	    "DB92_OP_Data".Msg_B0[16].%X1 := "DB114_MW_Meld".Ablauf_DF.Stoerung.GW_H;
	    "DB92_OP_Data".Msg_B0[16].%X2 := "DB114_MW_Meld".Ablauf_DF.Stoerung.GW_L;
	    "DB92_OP_Data".Msg_B0[16].%X3 := "DB114_MW_Meld".Ablauf_DF.Stoerung.GW_LL;
	    "DB92_OP_Data".Msg_B0[16].%X4 := "DB114_MW_Meld".Ablauf_pH.Stoerung.GW_HH;
	    "DB92_OP_Data".Msg_B0[16].%X5 := "DB114_MW_Meld".Ablauf_pH.Stoerung.GW_H;
	    "DB92_OP_Data".Msg_B0[16].%X6 := "DB114_MW_Meld".Ablauf_pH.Stoerung.GW_L;
	    "DB92_OP_Data".Msg_B0[16].%X7 := "DB114_MW_Meld".Ablauf_pH.Stoerung.GW_LL;
	    "DB92_OP_Data".Msg_B0[16].%X8 := "DB114_MW_Meld".Ablauf_O2.Stoerung.GW_HH;
	    "DB92_OP_Data".Msg_B0[16].%X9 := "DB114_MW_Meld".Ablauf_O2.Stoerung.GW_H;
	    "DB92_OP_Data".Msg_B0[16].%X10 := "DB114_MW_Meld".Ablauf_O2.Stoerung.GW_L;
	    "DB92_OP_Data".Msg_B0[16].%X11 := "DB114_MW_Meld".Ablauf_O2.Stoerung.GW_LL;
	    "DB92_OP_Data".Msg_B0[16].%X12 := "DB114_MW_Meld".Ablauf_Temp.Stoerung.GW_HH;
	    "DB92_OP_Data".Msg_B0[16].%X13 := "DB114_MW_Meld".Ablauf_Temp.Stoerung.GW_H;
	    "DB92_OP_Data".Msg_B0[16].%X14 := "DB114_MW_Meld".Ablauf_Temp.Stoerung.GW_L;
	    "DB92_OP_Data".Msg_B0[16].%X15 := "DB114_MW_Meld".Ablauf_Temp.Stoerung.GW_LL;
	    "DB92_OP_Data".Msg_B0[17].%X0 := "DB114_MW_Meld".Schlamm_ED_Niv.Stoerung.GW_HH;
	    "DB92_OP_Data".Msg_B0[17].%X1 := "DB114_MW_Meld".Schlamm_ED_Niv.Stoerung.GW_H;
	    "DB92_OP_Data".Msg_B0[17].%X2 := "DB114_MW_Meld".Schlamm_ED_Niv.Stoerung.GW_L;
	    "DB92_OP_Data".Msg_B0[17].%X3 := "DB114_MW_Meld".Schlamm_ED_Niv.Stoerung.GW_LL;
	    "DB92_OP_Data".Msg_B0[17].%X4 := "DB114_MW_Meld".Schlamm_Besch_Niv.Stoerung.GW_HH;
	    "DB92_OP_Data".Msg_B0[17].%X5 := "DB114_MW_Meld".Schlamm_Besch_Niv.Stoerung.GW_H;
	    "DB92_OP_Data".Msg_B0[17].%X6 := "DB114_MW_Meld".Schlamm_Besch_Niv.Stoerung.GW_L;
	    "DB92_OP_Data".Msg_B0[17].%X7 := "DB114_MW_Meld".Schlamm_Besch_Niv.Stoerung.GW_LL;
	    "DB92_OP_Data".Msg_B0[17].%X8 := "DB114_MW_Meld".Schlamm_Besch_DF.Stoerung.GW_HH;
	    "DB92_OP_Data".Msg_B0[17].%X9 := "DB114_MW_Meld".Schlamm_Besch_DF.Stoerung.GW_H;
	    "DB92_OP_Data".Msg_B0[17].%X10 := "DB114_MW_Meld".Schlamm_Besch_DF.Stoerung.GW_L;
	    "DB92_OP_Data".Msg_B0[17].%X11 := "DB114_MW_Meld".Schlamm_Besch_DF.Stoerung.GW_LL;
	    "DB92_OP_Data".Msg_B0[17].%X12 := "DB114_MW_Meld".Truebwasser_Niv.Stoerung.GW_HH;
	    "DB92_OP_Data".Msg_B0[17].%X13 := "DB114_MW_Meld".Truebwasser_Niv.Stoerung.GW_H;
	    "DB92_OP_Data".Msg_B0[17].%X14 := "DB114_MW_Meld".Truebwasser_Niv.Stoerung.GW_L;
	    "DB92_OP_Data".Msg_B0[17].%X15 := "DB114_MW_Meld".Truebwasser_Niv.Stoerung.GW_LL;
	    "DB92_OP_Data".Msg_B0[18].%X0 := "DB114_MW_Meld".Truebwasser_DF.Stoerung.GW_HH;
	    "DB92_OP_Data".Msg_B0[18].%X1 := "DB114_MW_Meld".Truebwasser_DF.Stoerung.GW_H;
	    "DB92_OP_Data".Msg_B0[18].%X2 := "DB114_MW_Meld".Truebwasser_DF.Stoerung.GW_L;
	    "DB92_OP_Data".Msg_B0[18].%X3 := "DB114_MW_Meld".Truebwasser_DF.Stoerung.GW_LL;
	    "DB92_OP_Data".Msg_B0[18].%X4 := "DB114_MW_Meld".Zulauf_SF_Niv.Stoerung.GW_HH;
	    "DB92_OP_Data".Msg_B0[18].%X5 := "DB114_MW_Meld".Zulauf_SF_Niv.Stoerung.GW_H;
	    "DB92_OP_Data".Msg_B0[18].%X6 := "DB114_MW_Meld".Zulauf_SF_Niv.Stoerung.GW_L;
	    "DB92_OP_Data".Msg_B0[18].%X7 := "DB114_MW_Meld".Zulauf_SF_Niv.Stoerung.GW_LL;
	    "DB92_OP_Data".Msg_B0[18].%X8 := "DB118_PW_Meld".FW_APW_Oeb_KB.Status.FWA_St;
	    "DB92_OP_Data".Msg_B0[18].%X9 := "DB118_PW_Meld".FW_APW_Oeb_KB.Status.FWA_P_St;
	    "DB92_OP_Data".Msg_B0[18].%X10 := "DB118_PW_Meld".FW_APW_Oeb_KB.Status.FWA_Ausf1;
	    "DB92_OP_Data".Msg_B0[18].%X11 := "DB118_PW_Meld".FW_APW_Oeb_KB.Status.FWA_Ausf2;
	    "DB92_OP_Data".Msg_B0[18].%X12 := "DB118_PW_Meld".FW_APW_Oeb_KB.Status.FWA_P1_St;
	    "DB92_OP_Data".Msg_B0[18].%X13 := "DB118_PW_Meld".FW_APW_Oeb_KB.Status.FWA_P2_St;
	    "DB92_OP_Data".Msg_B0[18].%X14 := "DB118_PW_Meld".FW_APW_Oeb_KB.Status.FWA_Niv_max;
	    "DB92_OP_Data".Msg_B0[18].%X15 := "DB118_PW_Meld".FW_APW_Oeb_KB.Status.FWA_EA_St;
	    "DB92_OP_Data".Msg_B0[19].%X0 := "DB118_PW_Meld".FW_APW_Oeb_KB.Status.Kom_St;
	    "DB92_OP_Data".Msg_B0[19].%X1 := "DB118_PW_Meld".FW_APW_Oeb_KB.Status.MW_Niv_St;
	    "DB92_OP_Data".Msg_B0[19].%X2 := "DB118_PW_Meld".FW_APW_Oeb_KB.Status.MW_DF_St;
	    "DB92_OP_Data".Msg_B0[19].%X3 := "DB118_PW_Meld".FW_APW_Oeb_KB.Status.MW_Dr_St;
	    "DB92_OP_Data".Msg_B0[19].%X4 := "DB118_PW_Meld".FW_APW_Oeb_KB.Status.MW_Res_St;
	    "DB92_OP_Data".Msg_B0[19].%X5 := "DB118_PW_Meld".FW_APW_BrR_DM.Status.FWA_St;
	    "DB92_OP_Data".Msg_B0[19].%X6 := "DB118_PW_Meld".FW_APW_BrR_DM.Status.FWA_P_St;
	    "DB92_OP_Data".Msg_B0[19].%X7 := "DB118_PW_Meld".FW_APW_BrR_DM.Status.FWA_Ausf1;
	    "DB92_OP_Data".Msg_B0[19].%X8 := "DB118_PW_Meld".FW_APW_BrR_DM.Status.FWA_Ausf2;
	    "DB92_OP_Data".Msg_B0[19].%X9 := "DB118_PW_Meld".FW_APW_BrR_DM.Status.FWA_P1_St;
	    "DB92_OP_Data".Msg_B0[19].%X10 := "DB118_PW_Meld".FW_APW_BrR_DM.Status.FWA_P2_St;
	    "DB92_OP_Data".Msg_B0[19].%X11 := "DB118_PW_Meld".FW_APW_BrR_DM.Status.FWA_Niv_max;
	    "DB92_OP_Data".Msg_B0[19].%X12 := "DB118_PW_Meld".FW_APW_BrR_DM.Status.FWA_EA_St;
	    "DB92_OP_Data".Msg_B0[19].%X13 := "DB118_PW_Meld".FW_APW_BrR_DM.Status.Kom_St;
	    "DB92_OP_Data".Msg_B0[19].%X14 := "DB118_PW_Meld".FW_APW_BrR_DM.Status.MW_Niv_St;
	    "DB92_OP_Data".Msg_B0[19].%X15 := "DB118_PW_Meld".FW_APW_BrR_DM.Status.MW_DF_St;
	    "DB92_OP_Data".Msg_B0[20].%X0 := "DB118_PW_Meld".FW_APW_BrR_DM.Status.MW_Dr_St;
	    "DB92_OP_Data".Msg_B0[20].%X1 := "DB118_PW_Meld".FW_APW_BrR_DM.Status.MW_Res_St;
	    "DB92_OP_Data".Msg_B0[20].%X2 := "DB118_PW_Meld".FW_APW_Oeb_Tu.Status.FWA_St;
	    "DB92_OP_Data".Msg_B0[20].%X3 := "DB118_PW_Meld".FW_APW_Oeb_Tu.Status.FWA_P_St;
	    "DB92_OP_Data".Msg_B0[20].%X4 := "DB118_PW_Meld".FW_APW_Oeb_Tu.Status.FWA_Ausf1;
	    "DB92_OP_Data".Msg_B0[20].%X5 := "DB118_PW_Meld".FW_APW_Oeb_Tu.Status.FWA_Ausf2;
	    "DB92_OP_Data".Msg_B0[20].%X6 := "DB118_PW_Meld".FW_APW_Oeb_Tu.Status.FWA_P1_St;
	    "DB92_OP_Data".Msg_B0[20].%X7 := "DB118_PW_Meld".FW_APW_Oeb_Tu.Status.FWA_P2_St;
	    "DB92_OP_Data".Msg_B0[20].%X8 := "DB118_PW_Meld".FW_APW_Oeb_Tu.Status.FWA_Niv_max;
	    "DB92_OP_Data".Msg_B0[20].%X9 := "DB118_PW_Meld".FW_APW_Oeb_Tu.Status.FWA_EA_St;
	    "DB92_OP_Data".Msg_B0[20].%X10 := "DB118_PW_Meld".FW_APW_Oeb_Tu.Status.Kom_St;
	    "DB92_OP_Data".Msg_B0[20].%X11 := "DB118_PW_Meld".FW_APW_Oeb_Tu.Status.MW_Niv_St;
	    "DB92_OP_Data".Msg_B0[20].%X12 := "DB118_PW_Meld".FW_APW_Oeb_Tu.Status.MW_DF_St;
	    "DB92_OP_Data".Msg_B0[20].%X13 := "DB118_PW_Meld".FW_APW_Oeb_Tu.Status.MW_Dr_St;
	    "DB92_OP_Data".Msg_B0[20].%X14 := "DB118_PW_Meld".FW_APW_Oeb_Tu.Status.MW_Res_St;
	    "DB92_OP_Data".Msg_B0[20].%X15 := "DB118_PW_Meld".FW_APW_Oeb_KS.Status.FWA_St;
	    "DB92_OP_Data".Msg_B0[21].%X0 := "DB118_PW_Meld".FW_APW_Oeb_KS.Status.FWA_P_St;
	    "DB92_OP_Data".Msg_B0[21].%X1 := "DB118_PW_Meld".FW_APW_Oeb_KS.Status.FWA_Ausf1;
	    "DB92_OP_Data".Msg_B0[21].%X2 := "DB118_PW_Meld".FW_APW_Oeb_KS.Status.FWA_Ausf2;
	    "DB92_OP_Data".Msg_B0[21].%X3 := "DB118_PW_Meld".FW_APW_Oeb_KS.Status.FWA_P1_St;
	    "DB92_OP_Data".Msg_B0[21].%X4 := "DB118_PW_Meld".FW_APW_Oeb_KS.Status.FWA_P2_St;
	    "DB92_OP_Data".Msg_B0[21].%X5 := "DB118_PW_Meld".FW_APW_Oeb_KS.Status.FWA_Niv_max;
	    "DB92_OP_Data".Msg_B0[21].%X6 := "DB118_PW_Meld".FW_APW_Oeb_KS.Status.FWA_EA_St;
	    "DB92_OP_Data".Msg_B0[21].%X7 := "DB118_PW_Meld".FW_APW_Oeb_KS.Status.Kom_St;
	    "DB92_OP_Data".Msg_B0[21].%X8 := "DB118_PW_Meld".FW_APW_Oeb_KS.Status.MW_Niv_St;
	    "DB92_OP_Data".Msg_B0[21].%X9 := "DB118_PW_Meld".FW_APW_Oeb_KS.Status.MW_DF_St;
	    "DB92_OP_Data".Msg_B0[21].%X10 := "DB118_PW_Meld".FW_APW_Oeb_KS.Status.MW_Dr_St;
	    "DB92_OP_Data".Msg_B0[21].%X11 := "DB118_PW_Meld".FW_APW_Oeb_KS.Status.MW_Res_St;
	    "DB92_OP_Data".Msg_B0[21].%X12 := "DB118_PW_Meld".FW_APW_Oeb_PG.Status.FWA_St;
	    "DB92_OP_Data".Msg_B0[21].%X13 := "DB118_PW_Meld".FW_APW_Oeb_PG.Status.FWA_P_St;
	    "DB92_OP_Data".Msg_B0[21].%X14 := "DB118_PW_Meld".FW_APW_Oeb_PG.Status.FWA_Ausf1;
	    "DB92_OP_Data".Msg_B0[21].%X15 := "DB118_PW_Meld".FW_APW_Oeb_PG.Status.FWA_Ausf2;
	    "DB92_OP_Data".Msg_B0[22].%X0 := "DB118_PW_Meld".FW_APW_Oeb_PG.Status.FWA_P1_St;
	    "DB92_OP_Data".Msg_B0[22].%X1 := "DB118_PW_Meld".FW_APW_Oeb_PG.Status.FWA_P2_St;
	    "DB92_OP_Data".Msg_B0[22].%X2 := "DB118_PW_Meld".FW_APW_Oeb_PG.Status.FWA_Niv_max;
	    "DB92_OP_Data".Msg_B0[22].%X3 := "DB118_PW_Meld".FW_APW_Oeb_PG.Status.FWA_EA_St;
	    "DB92_OP_Data".Msg_B0[22].%X4 := "DB118_PW_Meld".FW_APW_Oeb_PG.Status.Kom_St;
	    "DB92_OP_Data".Msg_B0[22].%X5 := "DB118_PW_Meld".FW_APW_Oeb_PG.Status.MW_Niv_St;
	    "DB92_OP_Data".Msg_B0[22].%X6 := "DB118_PW_Meld".FW_APW_Oeb_PG.Status.MW_DF_St;
	    "DB92_OP_Data".Msg_B0[22].%X7 := "DB118_PW_Meld".FW_APW_Oeb_PG.Status.MW_Dr_St;
	    "DB92_OP_Data".Msg_B0[22].%X8 := "DB118_PW_Meld".FW_APW_Oeb_PG.Status.MW_Res_St;
	    "DB92_OP_Data".Msg_B0[22].%X9 := "DB118_PW_Meld".FW_APW_Oeb_LW.Status.FWA_St;
	    "DB92_OP_Data".Msg_B0[22].%X10 := "DB118_PW_Meld".FW_APW_Oeb_LW.Status.FWA_P_St;
	    "DB92_OP_Data".Msg_B0[22].%X11 := "DB118_PW_Meld".FW_APW_Oeb_LW.Status.FWA_Ausf1;
	    "DB92_OP_Data".Msg_B0[22].%X12 := "DB118_PW_Meld".FW_APW_Oeb_LW.Status.FWA_Ausf2;
	    "DB92_OP_Data".Msg_B0[22].%X13 := "DB118_PW_Meld".FW_APW_Oeb_LW.Status.FWA_P1_St;
	    "DB92_OP_Data".Msg_B0[22].%X14 := "DB118_PW_Meld".FW_APW_Oeb_LW.Status.FWA_P2_St;
	    "DB92_OP_Data".Msg_B0[22].%X15 := "DB118_PW_Meld".FW_APW_Oeb_LW.Status.FWA_Niv_max;
	    "DB92_OP_Data".Msg_B0[23].%X0 := "DB118_PW_Meld".FW_APW_Oeb_LW.Status.FWA_EA_St;
	    "DB92_OP_Data".Msg_B0[23].%X1 := "DB118_PW_Meld".FW_APW_Oeb_LW.Status.Kom_St;
	    "DB92_OP_Data".Msg_B0[23].%X2 := "DB118_PW_Meld".FW_APW_Oeb_LW.Status.MW_Niv_St;
	    "DB92_OP_Data".Msg_B0[23].%X3 := "DB118_PW_Meld".FW_APW_Oeb_LW.Status.MW_DF_St;
	    "DB92_OP_Data".Msg_B0[23].%X4 := "DB118_PW_Meld".FW_APW_Oeb_LW.Status.MW_Dr_St;
	    "DB92_OP_Data".Msg_B0[23].%X5 := "DB118_PW_Meld".FW_APW_Oeb_LW.Status.MW_Res_St;
	    "DB92_OP_Data".Msg_B0[23].%X6 := "DB118_PW_Meld".FW_APW_GeD_WG.Status.FWA_St;
	    "DB92_OP_Data".Msg_B0[23].%X7 := "DB118_PW_Meld".FW_APW_GeD_WG.Status.FWA_P_St;
	    "DB92_OP_Data".Msg_B0[23].%X8 := "DB118_PW_Meld".FW_APW_GeD_WG.Status.FWA_Ausf1;
	    "DB92_OP_Data".Msg_B0[23].%X9 := "DB118_PW_Meld".FW_APW_GeD_WG.Status.FWA_Ausf2;
	    "DB92_OP_Data".Msg_B0[23].%X10 := "DB118_PW_Meld".FW_APW_GeD_WG.Status.FWA_P1_St;
	    "DB92_OP_Data".Msg_B0[23].%X11 := "DB118_PW_Meld".FW_APW_GeD_WG.Status.FWA_P2_St;
	    "DB92_OP_Data".Msg_B0[23].%X12 := "DB118_PW_Meld".FW_APW_GeD_WG.Status.FWA_Niv_max;
	    "DB92_OP_Data".Msg_B0[23].%X13 := "DB118_PW_Meld".FW_APW_GeD_WG.Status.FWA_EA_St;
	    "DB92_OP_Data".Msg_B0[23].%X14 := "DB118_PW_Meld".FW_APW_GeD_WG.Status.Kom_St;
	    "DB92_OP_Data".Msg_B0[23].%X15 := "DB118_PW_Meld".FW_APW_GeD_WG.Status.MW_Niv_St;
	    "DB92_OP_Data".Msg_B0[24].%X0 := "DB118_PW_Meld".FW_APW_GeD_WG.Status.MW_DF_St;
	    "DB92_OP_Data".Msg_B0[24].%X1 := "DB118_PW_Meld".FW_APW_GeD_WG.Status.MW_Dr_St;
	    "DB92_OP_Data".Msg_B0[24].%X2 := "DB118_PW_Meld".FW_APW_GeD_WG.Status.MW_Res_St;
	    "DB92_OP_Data".Msg_B0[24].%X3 := "DB118_PW_Meld".FW_APW_GeD_AA.Status.FWA_St;
	    "DB92_OP_Data".Msg_B0[24].%X4 := "DB118_PW_Meld".FW_APW_GeD_AA.Status.FWA_P_St;
	    "DB92_OP_Data".Msg_B0[24].%X5 := "DB118_PW_Meld".FW_APW_GeD_AA.Status.FWA_Ausf1;
	    "DB92_OP_Data".Msg_B0[24].%X6 := "DB118_PW_Meld".FW_APW_GeD_AA.Status.FWA_Ausf2;
	    "DB92_OP_Data".Msg_B0[24].%X7 := "DB118_PW_Meld".FW_APW_GeD_AA.Status.FWA_P1_St;
	    "DB92_OP_Data".Msg_B0[24].%X8 := "DB118_PW_Meld".FW_APW_GeD_AA.Status.FWA_P2_St;
	    "DB92_OP_Data".Msg_B0[24].%X9 := "DB118_PW_Meld".FW_APW_GeD_AA.Status.FWA_Niv_max;
	    "DB92_OP_Data".Msg_B0[24].%X10 := "DB118_PW_Meld".FW_APW_GeD_AA.Status.FWA_EA_St;
	    "DB92_OP_Data".Msg_B0[24].%X11 := "DB118_PW_Meld".FW_APW_GeD_AA.Status.Kom_St;
	    "DB92_OP_Data".Msg_B0[24].%X12 := "DB118_PW_Meld".FW_APW_GeD_AA.Status.MW_Niv_St;
	    "DB92_OP_Data".Msg_B0[24].%X13 := "DB118_PW_Meld".FW_APW_GeD_AA.Status.MW_DF_St;
	    "DB92_OP_Data".Msg_B0[24].%X14 := "DB118_PW_Meld".FW_APW_GeD_AA.Status.MW_Dr_St;
	    "DB92_OP_Data".Msg_B0[24].%X15 := "DB118_PW_Meld".FW_APW_GeD_AA.Status.MW_Res_St;
	    "DB92_OP_Data".Msg_B0[25].%X0 := "DB118_PW_Meld".FW_APW_WaD.Status.FWA_St;
	    "DB92_OP_Data".Msg_B0[25].%X1 := "DB118_PW_Meld".FW_APW_WaD.Status.FWA_P_St;
	    "DB92_OP_Data".Msg_B0[25].%X2 := "DB118_PW_Meld".FW_APW_WaD.Status.FWA_Ausf1;
	    "DB92_OP_Data".Msg_B0[25].%X3 := "DB118_PW_Meld".FW_APW_WaD.Status.FWA_Ausf2;
	    "DB92_OP_Data".Msg_B0[25].%X4 := "DB118_PW_Meld".FW_APW_WaD.Status.FWA_P1_St;
	    "DB92_OP_Data".Msg_B0[25].%X5 := "DB118_PW_Meld".FW_APW_WaD.Status.FWA_P2_St;
	    "DB92_OP_Data".Msg_B0[25].%X6 := "DB118_PW_Meld".FW_APW_WaD.Status.FWA_Niv_max;
	    "DB92_OP_Data".Msg_B0[25].%X7 := "DB118_PW_Meld".FW_APW_WaD.Status.FWA_EA_St;
	    "DB92_OP_Data".Msg_B0[25].%X8 := "DB118_PW_Meld".FW_APW_WaD.Status.Kom_St;
	    "DB92_OP_Data".Msg_B0[25].%X9 := "DB118_PW_Meld".FW_APW_WaD.Status.MW_Niv_St;
	    "DB92_OP_Data".Msg_B0[25].%X10 := "DB118_PW_Meld".FW_APW_WaD.Status.MW_DF_St;
	    "DB92_OP_Data".Msg_B0[25].%X11 := "DB118_PW_Meld".FW_APW_WaD.Status.MW_Dr_St;
	    "DB92_OP_Data".Msg_B0[25].%X12 := "DB118_PW_Meld".FW_APW_WaD.Status.MW_Res_St;
	    "DB92_OP_Data".Msg_B0[25].%X13 := "DB118_PW_Meld".FW_APW_WeD.Status.FWA_St;
	    "DB92_OP_Data".Msg_B0[25].%X14 := "DB118_PW_Meld".FW_APW_WeD.Status.FWA_P_St;
	    "DB92_OP_Data".Msg_B0[25].%X15 := "DB118_PW_Meld".FW_APW_WeD.Status.FWA_Ausf1;
	    "DB92_OP_Data".Msg_B0[26].%X0 := "DB118_PW_Meld".FW_APW_WeD.Status.FWA_Ausf2;
	    "DB92_OP_Data".Msg_B0[26].%X1 := "DB118_PW_Meld".FW_APW_WeD.Status.FWA_P1_St;
	    "DB92_OP_Data".Msg_B0[26].%X2 := "DB118_PW_Meld".FW_APW_WeD.Status.FWA_P2_St;
	    "DB92_OP_Data".Msg_B0[26].%X3 := "DB118_PW_Meld".FW_APW_WeD.Status.FWA_Niv_max;
	    "DB92_OP_Data".Msg_B0[26].%X4 := "DB118_PW_Meld".FW_APW_WeD.Status.FWA_EA_St;
	    "DB92_OP_Data".Msg_B0[26].%X5 := "DB118_PW_Meld".FW_APW_WeD.Status.Kom_St;
	    "DB92_OP_Data".Msg_B0[26].%X6 := "DB118_PW_Meld".FW_APW_WeD.Status.MW_Niv_St;
	    "DB92_OP_Data".Msg_B0[26].%X7 := "DB118_PW_Meld".FW_APW_WeD.Status.MW_DF_St;
	    "DB92_OP_Data".Msg_B0[26].%X8 := "DB118_PW_Meld".FW_APW_WeD.Status.MW_Dr_St;
	    "DB92_OP_Data".Msg_B0[26].%X9 := "DB118_PW_Meld".FW_APW_WeD.Status.MW_Res_St;
	    "DB92_OP_Data".Msg_B0[26].%X10 := "DB118_PW_Meld".FW_APW_NiD.Status.FWA_St;
	    "DB92_OP_Data".Msg_B0[26].%X11 := "DB118_PW_Meld".FW_APW_NiD.Status.FWA_P_St;
	    "DB92_OP_Data".Msg_B0[26].%X12 := "DB118_PW_Meld".FW_APW_NiD.Status.FWA_Ausf1;
	    "DB92_OP_Data".Msg_B0[26].%X13 := "DB118_PW_Meld".FW_APW_NiD.Status.FWA_Ausf2;
	    "DB92_OP_Data".Msg_B0[26].%X14 := "DB118_PW_Meld".FW_APW_NiD.Status.FWA_P1_St;
	    "DB92_OP_Data".Msg_B0[26].%X15 := "DB118_PW_Meld".FW_APW_NiD.Status.FWA_P2_St;
	    "DB92_OP_Data".Msg_B0[27].%X0 := "DB118_PW_Meld".FW_APW_NiD.Status.FWA_Niv_max;
	    "DB92_OP_Data".Msg_B0[27].%X1 := "DB118_PW_Meld".FW_APW_NiD.Status.FWA_EA_St;
	    "DB92_OP_Data".Msg_B0[27].%X2 := "DB118_PW_Meld".FW_APW_NiD.Status.Kom_St;
	    "DB92_OP_Data".Msg_B0[27].%X3 := "DB118_PW_Meld".FW_APW_NiD.Status.MW_Niv_St;
	    "DB92_OP_Data".Msg_B0[27].%X4 := "DB118_PW_Meld".FW_APW_NiD.Status.MW_DF_St;
	    "DB92_OP_Data".Msg_B0[27].%X5 := "DB118_PW_Meld".FW_APW_NiD.Status.MW_Dr_St;
	    "DB92_OP_Data".Msg_B0[27].%X6 := "DB118_PW_Meld".FW_APW_NiD.Status.MW_Res_St;
	    "DB92_OP_Data".Msg_B0[27].%X7 := "DB118_PW_Meld".FW_APW_LoS.Status.FWA_St;
	    "DB92_OP_Data".Msg_B0[27].%X8 := "DB118_PW_Meld".FW_APW_LoS.Status.FWA_P_St;
	    "DB92_OP_Data".Msg_B0[27].%X9 := "DB118_PW_Meld".FW_APW_LoS.Status.FWA_Ausf1;
	    "DB92_OP_Data".Msg_B0[27].%X10 := "DB118_PW_Meld".FW_APW_LoS.Status.FWA_Ausf2;
	    "DB92_OP_Data".Msg_B0[27].%X11 := "DB118_PW_Meld".FW_APW_LoS.Status.FWA_P1_St;
	    "DB92_OP_Data".Msg_B0[27].%X12 := "DB118_PW_Meld".FW_APW_LoS.Status.FWA_P2_St;
	    "DB92_OP_Data".Msg_B0[27].%X13 := "DB118_PW_Meld".FW_APW_LoS.Status.FWA_Niv_max;
	    "DB92_OP_Data".Msg_B0[27].%X14 := "DB118_PW_Meld".FW_APW_LoS.Status.FWA_EA_St;
	    "DB92_OP_Data".Msg_B0[27].%X15 := "DB118_PW_Meld".FW_APW_LoS.Status.Kom_St;
	    "DB92_OP_Data".Msg_B0[28].%X0 := "DB118_PW_Meld".FW_APW_LoS.Status.MW_Niv_St;
	    "DB92_OP_Data".Msg_B0[28].%X1 := "DB118_PW_Meld".FW_APW_LoS.Status.MW_DF_St;
	    "DB92_OP_Data".Msg_B0[28].%X2 := "DB118_PW_Meld".FW_APW_LoS.Status.MW_Dr_St;
	    "DB92_OP_Data".Msg_B0[28].%X3 := "DB118_PW_Meld".FW_APW_LoS.Status.MW_Res_St;
	    "DB92_OP_Data".Msg_B0[28].%X4 := "DB118_PW_Meld".FW_APW_Oeb_Ge.Status.FWA_St;
	    "DB92_OP_Data".Msg_B0[28].%X5 := "DB118_PW_Meld".FW_APW_Oeb_Ge.Status.FWA_P_St;
	    "DB92_OP_Data".Msg_B0[28].%X6 := "DB118_PW_Meld".FW_APW_Oeb_Ge.Status.FWA_Ausf1;
	    "DB92_OP_Data".Msg_B0[28].%X7 := "DB118_PW_Meld".FW_APW_Oeb_Ge.Status.FWA_Ausf2;
	    "DB92_OP_Data".Msg_B0[28].%X8 := "DB118_PW_Meld".FW_APW_Oeb_Ge.Status.FWA_P1_St;
	    "DB92_OP_Data".Msg_B0[28].%X9 := "DB118_PW_Meld".FW_APW_Oeb_Ge.Status.FWA_P2_St;
	    "DB92_OP_Data".Msg_B0[28].%X10 := "DB118_PW_Meld".FW_APW_Oeb_Ge.Status.FWA_Niv_max;
	    "DB92_OP_Data".Msg_B0[28].%X11 := "DB118_PW_Meld".FW_APW_Oeb_Ge.Status.FWA_EA_St;
	    "DB92_OP_Data".Msg_B0[28].%X12 := "DB118_PW_Meld".FW_APW_Oeb_Ge.Status.Kom_St;
	    "DB92_OP_Data".Msg_B0[28].%X13 := "DB118_PW_Meld".FW_APW_Oeb_Ge.Status.MW_Niv_St;
	    "DB92_OP_Data".Msg_B0[28].%X14 := "DB118_PW_Meld".FW_APW_Oeb_Ge.Status.MW_DF_St;
	    "DB92_OP_Data".Msg_B0[28].%X15 := "DB118_PW_Meld".FW_APW_Oeb_Ge.Status.MW_Dr_St;
	    "DB92_OP_Data".Msg_B0[29].%X0 := "DB118_PW_Meld".FW_APW_Oeb_Ge.Status.MW_Res_St;
	    "DB92_OP_Data".Msg_B0[29].%X1 := "DB118_PW_Meld".FW_APW_BuH.Status.FWA_St;
	    "DB92_OP_Data".Msg_B0[29].%X2 := "DB118_PW_Meld".FW_APW_BuH.Status.FWA_P_St;
	    "DB92_OP_Data".Msg_B0[29].%X3 := "DB118_PW_Meld".FW_APW_BuH.Status.FWA_Ausf1;
	    "DB92_OP_Data".Msg_B0[29].%X4 := "DB118_PW_Meld".FW_APW_BuH.Status.FWA_Ausf2;
	    "DB92_OP_Data".Msg_B0[29].%X5 := "DB118_PW_Meld".FW_APW_BuH.Status.FWA_P1_St;
	    "DB92_OP_Data".Msg_B0[29].%X6 := "DB118_PW_Meld".FW_APW_BuH.Status.FWA_P2_St;
	    "DB92_OP_Data".Msg_B0[29].%X7 := "DB118_PW_Meld".FW_APW_BuH.Status.FWA_Niv_max;
	    "DB92_OP_Data".Msg_B0[29].%X8 := "DB118_PW_Meld".FW_APW_BuH.Status.FWA_EA_St;
	    "DB92_OP_Data".Msg_B0[29].%X9 := "DB118_PW_Meld".FW_APW_BuH.Status.Kom_St;
	    "DB92_OP_Data".Msg_B0[29].%X10 := "DB118_PW_Meld".FW_APW_BuH.Status.MW_Niv_St;
	    "DB92_OP_Data".Msg_B0[29].%X11 := "DB118_PW_Meld".FW_APW_BuH.Status.MW_DF_St;
	    "DB92_OP_Data".Msg_B0[29].%X12 := "DB118_PW_Meld".FW_APW_BuH.Status.MW_Dr_St;
	    "DB92_OP_Data".Msg_B0[29].%X13 := "DB118_PW_Meld".FW_APW_BuH.Status.MW_Res_St;
	    "DB92_OP_Data".Msg_B0[29].%X14 := "DB118_PW_Meld".FW_APW_BrR_TS.Status.FWA_St;
	    "DB92_OP_Data".Msg_B0[29].%X15 := "DB118_PW_Meld".FW_APW_BrR_TS.Status.FWA_P_St;
	    "DB92_OP_Data".Msg_B0[30].%X0 := "DB118_PW_Meld".FW_APW_BrR_TS.Status.FWA_Ausf1;
	    "DB92_OP_Data".Msg_B0[30].%X1 := "DB118_PW_Meld".FW_APW_BrR_TS.Status.FWA_Ausf2;
	    "DB92_OP_Data".Msg_B0[30].%X2 := "DB118_PW_Meld".FW_APW_BrR_TS.Status.FWA_P1_St;
	    "DB92_OP_Data".Msg_B0[30].%X3 := "DB118_PW_Meld".FW_APW_BrR_TS.Status.FWA_P2_St;
	    "DB92_OP_Data".Msg_B0[30].%X4 := "DB118_PW_Meld".FW_APW_BrR_TS.Status.FWA_Niv_max;
	    "DB92_OP_Data".Msg_B0[30].%X5 := "DB118_PW_Meld".FW_APW_BrR_TS.Status.FWA_EA_St;
	    "DB92_OP_Data".Msg_B0[30].%X6 := "DB118_PW_Meld".FW_APW_BrR_TS.Status.Kom_St;
	    "DB92_OP_Data".Msg_B0[30].%X7 := "DB118_PW_Meld".FW_APW_BrR_TS.Status.MW_Niv_St;
	    "DB92_OP_Data".Msg_B0[30].%X8 := "DB118_PW_Meld".FW_APW_BrR_TS.Status.MW_DF_St;
	    "DB92_OP_Data".Msg_B0[30].%X9 := "DB118_PW_Meld".FW_APW_BrR_TS.Status.MW_Dr_St;
	    "DB92_OP_Data".Msg_B0[30].%X10 := "DB118_PW_Meld".FW_APW_BrR_TS.Status.MW_Res_St;
	    "DB92_OP_Data".Msg_B0[30].%X11 := "DB104_Antriebe_Meld".BB1_SR_K.Stoerung.Wa_EZ;
	    "DB92_OP_Data".Msg_B0[30].%X12 := "DB104_Antriebe_Meld".BB1_SR_K.Stoerung.Wa_Wart;
	    "DB92_OP_Data".Msg_B0[30].%X13 := "DB104_Antriebe_Meld".BB2_SR_K.Stoerung.Wa_EZ;
	    "DB92_OP_Data".Msg_B0[30].%X14 := "DB104_Antriebe_Meld".BB2_SR_K.Stoerung.Wa_Wart;


	END_IF;


END_FUNCTION

FUNCTION "Allgemein" : Void
{ S7_Optimized_Access := 'TRUE' }
VERSION : 0.1
   VAR_TEMP
      retval : Int;
      b_tmp : Bool;
   END_VAR


BEGIN

	//Anlaufphase
	//

	IF "FirstScan" THEN
	    "SPS_Anlauf" := 0;
	    "DB92_OP_Data".SPS_Idx := "SPS_Idx_eigen";
	    "DB92_OP_Data".SPS_Idx_BitIdx := SHL(IN := BYTE#1, N := INT_TO_UINT("SPS_Idx_eigen"));
	END_IF;


	"FC61_TON_s"(enable:="SPS_Anlauf",
	           Imp:="Imp_Sek",
	           TmrMax:=5,
	           TmrVar:="Tmr_Anlauf_AG",
	           Q:=#b_tmp);

	IF #b_tmp THEN
	    "Wiederanlauf" := 1;
	END_IF;
	IF NOT "SPS_Anlauf" THEN
	    "Wiederanlauf_NA_chk" := 1;
	END_IF;

	//Ablauf nach Netzwiederkehr
	//Zuweisung setzen!!
	"Notstrombetrieb" := 0;
	"Netzausfall" := ( ("ZEN_Meld".E_NSHV_NA OR NOT "ZEN_Meld".E_NSHV_LS_Aus) AND NOT "Notstrombetrieb")AND FALSE;
	"ZEN_Meld".ZEN_NA_res := "Netzausfall";

	//nach Freigabe Peripherie Netzausfallsignal berücksichtigen
	#b_tmp := NOT "Netzausfall";

	"FC61_TON_s"(enable := #b_tmp,
	           Imp := "Imp_Sek",
	           TmrMax := 30,
	           TmrVar := "Tmr_Netzwiederkehr",
	           Q := #b_tmp);

	IF ("Freigabe_Peripherie" AND NOT "Netzausfall") OR #b_tmp THEN
	    "Freigabe_Verbraucher" := 1;
	END_IF;

	//Erzeugung globaler Quittierimpuls
	//
	//"UV_DEK_Bef".KAW_DEK_BF_Quit OR ("UV_DEK_Bef_UV".KAW_DEK_BF_Quit AND "UV_DEK_Meld".KAW_DEK_Bed_aktiv)
	//
	"FC62_TOF_s"(enable:="ZEN_Bef".ZEN_Quit_BF,
	             Imp:="Imp_Sek",
	             TmrMax:=2,
	             TmrVar:="Tmr_GlobalQuit",
	             Q:="Global_Quit");
	//Quittierung Meldesystem OP triggern
	"DB92_OP_Data".MsgQuit := (("ZEN_Bef".ZEN_Quit_BF) AND "ZEN_Meld".ZEN_Bed_aktiv);


	"ZEN_Bef".ZEN_Quit_BF := 0;


	//Uhrzeitverwaltung
	//

	"IDB_FB51_Time"();



	//Abfrage DP-Teilnehmer nach SPS-Anlauf

	"FC61_TON_s"(enable := "Wiederanlauf",
	           Imp := "Imp_Sek",
	           TmrMax := 2,
	           TmrVar := "Tmr_Freigabe_Peripherie",
	           Q := #b_tmp);
	IF #b_tmp THEN
	    "Freigabe_Peripherie" := 1;
	    "Freigabe_Zyklus" := 1;
	    #retval:=DeviceStates(LADDR := 259, MODE := 4, STATE := "DB91_DP_aktiv".Tln);
	END_IF;




END_FUNCTION

FUNCTION_BLOCK "FB55_PulsPause"
{ S7_Optimized_Access := 'TRUE' }
VERSION : 0.1
   VAR_INPUT
      enable { ExternalAccessible := 'False'; ExternalVisible := 'False'; ExternalWritable := 'False'} : Bool;
      Pulszeit { ExternalAccessible := 'False'; ExternalVisible := 'False'; ExternalWritable := 'False'} : DInt;
      Pausenzeit { ExternalAccessible := 'False'; ExternalVisible := 'False'; ExternalWritable := 'False'} : DInt;
   END_VAR

   VAR_OUTPUT
      Operation { ExternalAccessible := 'False'; ExternalVisible := 'False'; ExternalWritable := 'False'} : Bool;
   END_VAR

   VAR
      Tmr_Zt_Puls {InstructionName := 'TON_TIME'; LibVersion := '1.0'; ExternalAccessible := 'False'; ExternalVisible := 'False'; ExternalWritable := 'False'} : TON_TIME;
      Tmr_Zt_Pause {InstructionName := 'TON_TIME'; LibVersion := '1.0'; ExternalAccessible := 'False'; ExternalVisible := 'False'; ExternalWritable := 'False'} : TON_TIME;
      aktiv { ExternalAccessible := 'False'; ExternalVisible := 'False'; ExternalWritable := 'False'} : Bool;
      FM_init { ExternalAccessible := 'False'; ExternalVisible := 'False'; ExternalWritable := 'False'} : Bool;
   END_VAR


BEGIN

	IF #enable AND #Pulszeit>0 AND #Pausenzeit>0 THEN
	    IF NOT #aktiv AND NOT #Tmr_Zt_Pause.Q THEN
	        #aktiv := 1;
	    END_IF;
	ELSE
	    #aktiv := 0;
	END_IF;
	#FM_init := #enable;

	#Tmr_Zt_Puls(IN:=#aktiv,
	             PT:=DINT_TO_TIME(#Pulszeit*DINT#1000));

	#Tmr_Zt_Pause(IN := #Tmr_Zt_Puls.Q,
	              PT := DINT_TO_TIME(#Pausenzeit * DINT#1000));

	IF #Tmr_Zt_Pause.Q THEN
	    #aktiv := 0;
	END_IF;
	#Operation := (#aktiv AND NOT #Tmr_Zt_Puls.Q) OR (#enable AND (#Pausenzeit = 0));
END_FUNCTION_BLOCK

FUNCTION_BLOCK "FB59_Mittelwert_imp"
{ S7_Optimized_Access := 'TRUE' }
VERSION : 0.1
   VAR_INPUT
      Zeitfenster { ExternalAccessible := 'False'; ExternalVisible := 'False'; ExternalWritable := 'False'} : DInt := 60;
      Rohwert { ExternalAccessible := 'False'; ExternalVisible := 'False'; ExternalWritable := 'False'} : Real;
      Rohwert_nok { ExternalAccessible := 'False'; ExternalVisible := 'False'; ExternalWritable := 'False'} : Bool;
      Imp { ExternalAccessible := 'False'; ExternalVisible := 'False'; ExternalWritable := 'False'} : Bool;
   END_VAR

   VAR_OUTPUT
      Mittelwert { ExternalAccessible := 'False'; ExternalVisible := 'False'; ExternalWritable := 'False'} : Real;
   END_VAR

   VAR_IN_OUT
      MemDB : "T_MW_MITTEL";
   END_VAR

   VAR
      DataIdx_max { ExternalAccessible := 'False'; ExternalVisible := 'False'; ExternalWritable := 'False'} : Int;
      curInIdx { ExternalAccessible := 'False'; ExternalVisible := 'False'; ExternalWritable := 'False'} : Int;
      valid_Window { ExternalAccessible := 'False'; ExternalVisible := 'False'; ExternalWritable := 'False'} : Int;
   END_VAR

   VAR_TEMP
      i : Int;
      s : Real;
   END_VAR

   VAR CONSTANT
      MaxEntries : Int := 120;
   END_VAR


BEGIN
	    IF #Zeitfenster <= 0 THEN
	        #DataIdx_max := 0;
	    ELSIF #Zeitfenster > #MaxEntries THEN
	        #DataIdx_max := #MaxEntries - 1;
	    ELSE
	        #DataIdx_max := DINT_TO_INT(#Zeitfenster) - 1;
	    END_IF;
	    IF #Rohwert_nok OR #DataIdx_max = 0 THEN
	        #curInIdx := 0;
	        #valid_Window := 0;
	        #Mittelwert := #Rohwert;
	    ELSE

	        IF #Imp THEN
	            #MemDB.Values[#curInIdx] := #Rohwert;
	            #curInIdx := #curInIdx + 1;
	            IF #curInIdx > #DataIdx_max THEN
	                #curInIdx := 0;
	            END_IF;
	            #s := 0.0;
	            FOR #i := 0 TO #valid_Window DO
	                #s := #s + #MemDB.Values[#i];
	            END_FOR;
	            #Mittelwert := #s / (INT_TO_REAL(#valid_Window + 1));
	            IF #valid_Window < #DataIdx_max THEN
	                #valid_Window := #valid_Window + 1;
	            ELSE
	                #valid_Window := #DataIdx_max;
	            END_IF;
	        END_IF;
	    END_IF;

END_FUNCTION_BLOCK

ORGANIZATION_BLOCK "Main"
TITLE = "Main Program Sweep (Cycle)"
{ S7_Optimized_Access := 'TRUE' }
VERSION : 0.1

BEGIN


	"Allgemein"();
	"Peripherie"();

	IF "Freigabe_Zyklus" THEN

	    "FB1_Antriebe_IDB"();
	    "FB2_Messwerte_IDB"();
	    "FB3_Automatik_Belebung_IDB"();
	    "FB4_Automatik_Biocos_IDB"();
	    "FB5_Automatik_Zulauf_Ablauf_IDB"();


	    "FB6_Kommunikation_IDB"();
	    "FB7_Pumpwerke_IDB"();

	    "FB8_Leitstelle_IDB"();
	    "FB9_USV_Kom_IDB"();

	END_IF;


	"SPS_Anlauf" := 1;
END_ORGANIZATION_BLOCK

